Fanuc KAREL source: kc00020.KL

-- PROVISIONAL review KL for V770-1; original PC SHA256 2f295e2ab65331e97ee8f0c63d4a039e3dbfa9ac8707be9f56404de2bef6f488
-- Incomplete behavior may be omitted. Consult companion uncertainty JSON. Do not deploy.
PROGRAM KC00020
%NOLOCKGROUP
BEGIN
  -- UNRESOLVED_PC offsets 5-12; opcodes 27,27,27,9C,31
  -- UNRESOLVED_PC offsets 17-21; opcodes 7F
END KC00020
